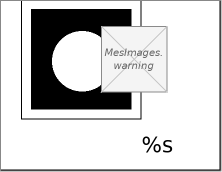
VISUALIZATION VISU_POMPE_TURBO  // 222x172
VAR_IN_OUT
	m_Input_POMPE : BLOCK_PPM_DEF;
END_VAR
    Rectangle (0,0 220x170), invisible if: TRUE
    Rectangle (96,130 123x30), "%s", text variable: m_Input_POMPE.MNEMO
    Rectangle (31,9 100x100), colour toggle: (m_Input_POMPE.OUT_ON) <> 0
    Rectangle (31,9 100x100), colour toggle: (m_Input_POMPE.STATE_ON) <> 0, invisible if: NOT m_Input_POMPE.STATE_ON AND NOT m_Input_POMPE.STATE_OFF
    Group (47,26 68x68)
        Ellipse (0,0 70x70)
        Polyline (65,36)
        Polyline (5,42)
        Polyline (15,42)
        Polyline (25,42)
        Polyline (35,42)
        Polyline (45,42)
        Polyline (55,42)
        Polyline (65,42)
    Rectangle (21,0 120x119), invisible if: NOT (m_Input_POMPE.Autor_ON_IHM OR m_Input_POMPE.Autor_OFF_IHM) OR NOT PRG_User.ACTU_USER.MAINTENANCE
        tap m_Input_POMPE.M_ON
    Image (101,26 66x66), invisible if: NOT m_Input_POMPE.STATE_NOK, image: MesImages.warning
END_VISUALIZATION

(* stored: Version 1.1.0.1, ProductVersion 3.1.4024.10
   Visu VISU_POMPE_TURBO: Id {54dffb44-694b-4e4a-ab3a-6b6f7e028e6e} *)
